TYPE DUT_Kamer :
STRUCT
    Licht : BOOL;
    Temperatuur : REAL;
    MA_Temp : REAL;
END_STRUCT
END_TYPE

(* stored: Version 1.1.0.1, ProductVersion 3.1.4024.15
   DUT DUT_Kamer: Id {1bfcf178-7c27-4a9b-a8a3-ef240f14cd6c} *)
